//==================================================================================================
//								RJM Maszyny sp. z o.o.
//									13.05.2022
//	Obsługa silonwika z zawrorem 5 na 3 - Zapowietrzony
//	Realizacja wysuwania i chowania tłoczyska dla jednej cewki zwrócenie pozycji skrajnych
// 	v1.0	|| TC v 3.1.4024.22		|| - pierwsza wersja
//==================================================================================================
FUNCTION_BLOCK FB_Silownik_5na3_Zapowietrzony EXTENDS FB_SIlownikBaza
VAR_INPUT
END_VAR
VAR_OUTPUT
END_VAR
VAR
	bCewkaB							AT %Q*	: BOOL;	
END_VAR

METHOD Praca : BOOL
VAR_INPUT
END_VAR
SUPER^.Praca ();

IF (bPrzesuwanieWStroneKonca AND NOT bCewkaA) THEN
	bCewkaB									:= TRUE;
END_IF
IF  (bPrzesuwanieWStronePoczatku AND bCewkaA) THEN
	bCewkaB									:= FALSE;
END_IF

IF (bPrzesuwanieWStronePoczatku AND NOT bCewkaB) THEN
	bCewkaA									:= TRUE;
END_IF
IF  (bPrzesuwanieWStroneKonca AND bCewkaB) THEN
	bCewkaA									:= FALSE;
END_IF
END_METHOD

END_FUNCTION_BLOCK

(* stored: Version 1.1.0.1, ProductVersion 3.1.4024.11
   POU FB_Silownik_5na3_Zapowietrzony: Id {689641be-6248-4354-8b1a-b73eaa308931}, SpecialFunc None
   Method Praca: Id {ab5c0f77-98f8-4d17-a110-76fe822a69fa} *)
